FUNCTION_BLOCK EQ_NeedleAxis (* Needle lift with down/up valves, end switches and a position sensor; owns its IO points; commands Stop=0, Down=1, Up=2 *)
  (* Standard: 61499-2 *)
  (* Version 0.1, 2026-09-28, Project contributors, AAU Smart Production Lab *)
  PACKAGE filler;
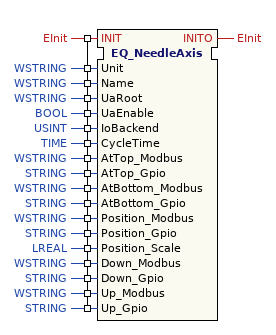
  EVENT_INPUT
    INIT : EInit WITH Unit, Name, UaRoot, UaEnable, IoBackend, CycleTime, AtTop_Modbus, AtTop_Gpio, AtBottom_Modbus, AtBottom_Gpio, Position_Modbus, Position_Gpio, Position_Scale, Down_Modbus, Down_Gpio, Up_Modbus, Up_Gpio;
  END_EVENT
  EVENT_OUTPUT
    INITO : EInit;
  END_EVENT
  VAR_INPUT
    Unit : WSTRING;
    Name : WSTRING := "NeedleAxis";
    UaRoot : WSTRING;
    UaEnable : BOOL;
    IoBackend : USINT := 2;
    CycleTime : TIME := T#50ms;
    AtTop_Modbus : WSTRING;
    AtTop_Gpio : STRING;
    AtBottom_Modbus : WSTRING;
    AtBottom_Gpio : STRING;
    Position_Modbus : WSTRING;
    Position_Gpio : STRING;
    Position_Scale : LREAL := 0.1;
    Down_Modbus : WSTRING;
    Down_Gpio : STRING;
    Up_Modbus : WSTRING;
    Up_Gpio : STRING;
  END_VAR
  FBS
    Logic : filler::EL_NeedleAxis;
    SubCmd : iec61499::net::SUBSCRIBE_1(QI := TRUE);
    PubState : iec61499::net::PUBLISH_3(QI := TRUE);
    PubUa : iec61499::net::PUBLISH_3;
    In_AtTop : unitlib::IO_DI;
    In_AtBottom : unitlib::IO_DI;
    In_Position : unitlib::IO_AI;
    Out_Down : unitlib::IO_DO;
    Out_Up : unitlib::IO_DO;
    Cycle : iec61499::events::E_CYCLE;
  END_FBS
  EVENT_CONNECTIONS
    INIT TO Logic.INIT;
    Logic.INITO TO SubCmd.INIT;
    SubCmd.INITO TO PubState.INIT;
    PubState.INITO TO PubUa.INIT;
    PubUa.INITO TO In_AtTop.INIT;
    In_AtTop.INITO TO In_AtBottom.INIT;
    In_AtBottom.INITO TO In_Position.INIT;
    In_Position.INITO TO Out_Down.INIT;
    Out_Down.INITO TO Out_Up.INIT;
    Out_Up.INITO TO Cycle.START;
    Out_Up.INITO TO INITO;
    SubCmd.IND TO Logic.CMD;
    Cycle.EO TO In_AtTop.REQ;
    In_AtTop.CNF TO In_AtBottom.REQ;
    In_AtBottom.CNF TO In_Position.REQ;
    In_Position.CNF TO Logic.SAMPLE;
    Logic.STATE TO PubState.REQ;
    Logic.STATE TO PubUa.REQ;
    Logic.DRIVE TO Out_Down.REQ;
    Out_Down.CNF TO Out_Up.REQ;
    Out_Up.CNF TO Logic.DRIVEN;
  END_CONNECTIONS
  DATA_CONNECTIONS
    Unit TO Logic.Unit;
    Name TO Logic.Name;
    UaRoot TO Logic.UaRoot;
    Logic.IdCmd TO SubCmd.ID;
    Logic.IdState TO PubState.ID;
    Logic.IdPub TO PubUa.ID;
    UaEnable TO PubUa.QI;
    CycleTime TO Cycle.DT;
    SubCmd.RD_1 TO Logic.Command;
    IoBackend TO In_AtTop.Backend;
    AtTop_Modbus TO In_AtTop.ModbusId;
    AtTop_Gpio TO In_AtTop.GpioName;
    In_AtTop.IN TO Logic.I_AtTop;
    Logic.AtTop TO PubState.SD_1;
    Logic.AtTop TO PubUa.SD_1;
    IoBackend TO In_AtBottom.Backend;
    AtBottom_Modbus TO In_AtBottom.ModbusId;
    AtBottom_Gpio TO In_AtBottom.GpioName;
    In_AtBottom.IN TO Logic.I_AtBottom;
    Logic.AtBottom TO PubState.SD_2;
    Logic.AtBottom TO PubUa.SD_2;
    IoBackend TO In_Position.Backend;
    Position_Modbus TO In_Position.ModbusId;
    Position_Gpio TO In_Position.GpioName;
    Position_Scale TO In_Position.Scale;
    In_Position.IN TO Logic.I_Position;
    Logic.Position TO PubState.SD_3;
    Logic.Position TO PubUa.SD_3;
    IoBackend TO Out_Down.Backend;
    Down_Modbus TO Out_Down.ModbusId;
    Down_Gpio TO Out_Down.GpioName;
    Logic.O_Down TO Out_Down.OUT;
    IoBackend TO Out_Up.Backend;
    Up_Modbus TO Out_Up.ModbusId;
    Up_Gpio TO Out_Up.GpioName;
    Logic.O_Up TO Out_Up.OUT;
  END_CONNECTIONS
END_FUNCTION_BLOCK
